(* CODESYS project HeatSealSequence.xml

Project tree, tasks and I/O mapping:
  function block HeatSealSequence [SFC]
*)

// HeatSealSequence
FUNCTION_BLOCK HeatSealSequence
VAR_INPUT
	SFCInit: BOOL; // Disable bit
	Open: BOOL; // Command open
	Close: BOOL; // Command close
	OpenSensor: BOOL; // Open sensor input
	CloseSensor: BOOL; // Close sensor input
	SFCReset: BOOL; // Stop bit
	Reset: BOOL;
END_VAR
VAR_OUTPUT
	Forward: BOOL; // Motor output forward
	Reverse: BOOL; // Motor output reverse
	Brake: BOOL; // Motor output brake activated
	Closed: BOOL;
	Opened: BOOL;
END_VAR
VAR
END_VAR

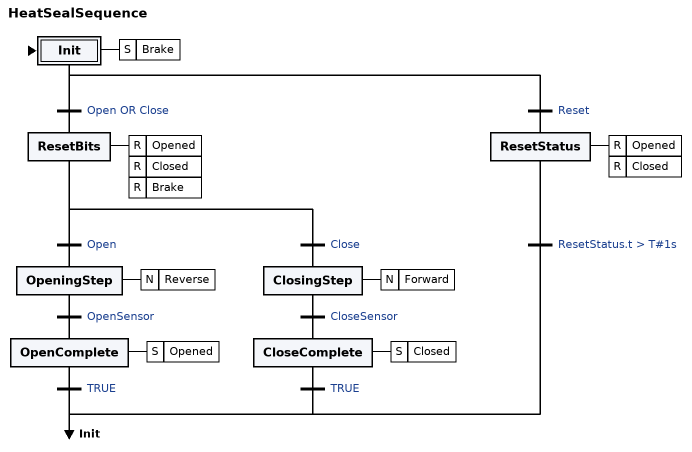
INITIAL_STEP Init:
    Brake(S);
END_STEP
TRANSITION FROM Init TO ResetBits
    := Open OR Close;
END_TRANSITION
STEP ResetBits:
    Opened(R);
    Closed(R);
    Brake(R);
END_STEP
TRANSITION FROM ResetBits TO OpeningStep
    := Open;
END_TRANSITION
STEP OpeningStep:
    Reverse(N);
END_STEP
TRANSITION FROM OpeningStep TO OpenComplete
    := OpenSensor;
END_TRANSITION
STEP OpenComplete:
    Opened(S);
END_STEP
TRANSITION FROM OpenComplete TO Init
    := TRUE;
END_TRANSITION
TRANSITION FROM ResetBits TO ClosingStep
    := Close;
END_TRANSITION
STEP ClosingStep:
    Forward(N);
END_STEP
TRANSITION FROM ClosingStep TO CloseComplete
    := CloseSensor;
END_TRANSITION
STEP CloseComplete:
    Closed(S);
END_STEP
TRANSITION FROM CloseComplete TO Init
    := TRUE;
END_TRANSITION
TRANSITION FROM Init TO ResetStatus
    := Reset;
END_TRANSITION
STEP ResetStatus:
    Opened(R);
    Closed(R);
END_STEP
TRANSITION FROM ResetStatus TO Init
    := ResetStatus.t > T#1s;
END_TRANSITION

END_FUNCTION_BLOCK
